INTERFACE IReadOnlyDictionary EXTENDS ICollection

METHOD ContainsGenericKey : BOOL
VAR_INPUT
	key : GENERIC_VALUE;
	releaseKey : BOOL := TRUE;
END_VAR
END_METHOD

METHOD ContainsKey : BOOL
VAR_INPUT
	key : ANY;
END_VAR
END_METHOD

// Negative value returned if not found
METHOD GetGenericKeyPosition : DINT
VAR_INPUT
	key : GENERIC_VALUE;
	releaseKey : BOOL := TRUE;
END_VAR
END_METHOD

// Negative value returned if not found
METHOD GetKeyPosition : DINT
VAR_INPUT
	key : ANY;
END_VAR
END_METHOD

METHOD GetKeyValuePairByIndex : REFERENCE TO GENERIC_KEY_VALUE_PAIR
VAR_INPUT
	index : DINT;
END_VAR
END_METHOD

METHOD TryGetValueByKey : BOOL
VAR_INPUT
	key : ANY;
END_VAR
VAR_OUTPUT
	value : GENERIC_VALUE;
END_VAR
END_METHOD

END_INTERFACE

(* stored: Version 1.1.0.1
   Itf IReadOnlyDictionary: Id {511d635b-9ee9-475d-b527-1b8927b91e7e}
   Method ContainsGenericKey: Id {9f8e7aad-b7e0-4834-94aa-20d7c5e1cdea}
   Method ContainsKey: Id {ff9cfb18-10ca-467e-9680-e293c6b611d5}
   Method GetGenericKeyPosition: Id {516cbd3d-5f27-4efd-8461-dc951eb682a7}
   Method GetKeyPosition: Id {5e2b0a29-a0f0-46ba-a9db-58fb22fe489f}
   Method GetKeyValuePairByIndex: Id {621d17f0-ce5c-4e12-9107-2706dfc65ad4}
   Method TryGetValueByKey: Id {c4542916-8eaf-41fb-a00c-f12b88d80700} *)
